{attribute 'qualified_only'}
{attribute 'strict'}
{attribute 'to_string'}
TYPE ST150_Cylinders_e : 
(
	Kraftbstutzung,
	_max
);
END_TYPE

(* stored: Version 1.1.0.1, ProductVersion 3.1.4024.6
   EnumerationTextList ST150_Cylinders_e: Id {88383a82-0561-4693-8192-ccab459a4427} *)
